// TwinCAT 3 PLC project Project1_1_PLC
// ProgramVersion: 3.1.4020.2
// libraries:
//   Tc2_Standard, * (Beckhoff Automation GmbH)
//   Tc2_System, * (Beckhoff Automation GmbH)
//   Tc3_Module, * (Beckhoff Automation GmbH)
// project tree:
//   / PlcTask.TcTTO
//   POUs/ POU.TcPOU

CONFIGURATION Project1_1_PLC
    RESOURCE PLC ON TwinCAT3
        TASK PlcTask(INTERVAL := T#10ms, PRIORITY := 20);
        PROGRAM POU WITH PlcTask : POU;
    END_RESOURCE
END_CONFIGURATION

// ---- POUs/POU.TcPOU
PROGRAM POU
VAR
	Container_in_place : BOOL;
	Container_full : BOOL;
	Tank_empty_in : BOOL;
	Loading : BOOL;
	Unloading : BOOL;
	Start : BOOL;
	Stop : BOOL;
	Emergency : BOOL;
	
	Motor : BOOL;
	Valve : BOOL;
	Tank_empty_out : BOOL;
	counter: INT;
	R_TRIG_0: R_TRIG;
END_VAR

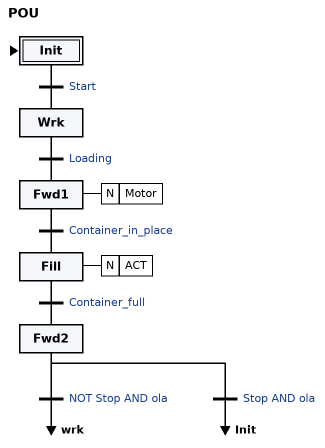
INITIAL_STEP Init:
END_STEP
TRANSITION FROM Init TO Wrk
    := Start;
END_TRANSITION
STEP Wrk:
END_STEP
TRANSITION FROM Wrk TO Fwd1
    := Loading;
END_TRANSITION
STEP Fwd1:
    Motor(N);
END_STEP
TRANSITION FROM Fwd1 TO Fill
    := Container_in_place;
END_TRANSITION
STEP Fill:
    ACT(N);
END_STEP
TRANSITION FROM Fill TO Fwd2
    := Container_full;
END_TRANSITION
STEP Fwd2:
END_STEP
TRANSITION FROM Fwd2 TO wrk
    := NOT Stop AND ola;
END_TRANSITION
TRANSITION FROM Fwd2 TO Init
    := Stop AND ola;
END_TRANSITION

ACTION ACT:
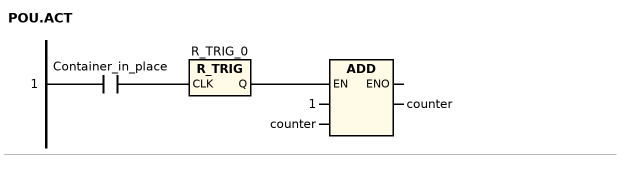
// NETWORK 1
R_TRIG_0(CLK := Container_in_place); // R_TRIG
IF R_TRIG_0.Q THEN counter := 1 + counter; END_IF
END_ACTION

TRANSITION ola:
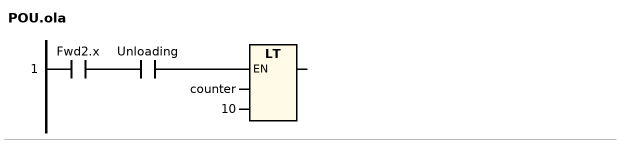
// NETWORK 1
(* Fwd2.x AND Unloading AND counter < 10; result not used *)
END_TRANSITION

END_PROGRAM
